// TIA Portal V16 export
// export: Created 2024-12-03T15:41:46.4557849Z, ExportSetting WithReadOnly, DisplayName Totally Integrated Automation Portal, DisplayVersion V16 Update 6, DisplayName TIA Portal Version Control Interface, DisplayVersion V16 Update 2, DisplayName TIA Portal Openness, DisplayVersion V16 Update 6, DisplayName TIA Portal Teamcenter Gateway, DisplayVersion V16, DisplayName SINAMICS Startdrive Advanced, DisplayVersion V16 Update 5, DisplayName SINAMICS Startdrive G130, G150, S120, S150, SINAMICS MV, S210, DisplayVersion V16 Update 5, DisplayName SINAMICS Startdrive G110M, G120, G120C, G120D, G120P, G115D, DisplayVersion V16 Update 5, DisplayName STEP 7 Professional, DisplayVersion V16 Update 6, DisplayName STEP 7 Safety, DisplayVersion V16, DisplayName WinCC Advanced / Unified PC, DisplayVersion V16 Update 6
TYPE "System_Counters_UDT"
// stored: CreationDate 2021-07-13T07:41:36.2278727Z, InterfaceModifiedDate 2021-03-11T07:33:04.7322472Z, IsConsistent true, LibraryConformanceStatus The object is library-conformant., ModifiedDate 2021-03-27T07:36:47.4918093Z
   STRUCT
      Infeed_1 : UInt;
      Infeed_2 : UInt;
      Infeed_3 : UInt;
      Infeed_4 : UInt;
      Infeed_5 : UInt;
      MainLane_Total : UInt;
      Scan100_Reject : UInt;
      Scan100_Exit1 : UInt;
      Scan100_Exit2 : UInt;
      Scan100MainLane : UInt;
      Scan200_Rejct : UInt;
      Scan200_Printer1 : UInt;
      Scan200_Printer2 : UInt;
      Scan200_Printer3 : UInt;
      Scan200_MainLane : UInt;
      MezzanineRetour_Printer1 : UInt;
      MezzanineRetour_Printer2 : UInt;
      Printer1_OK : UInt;
      Printer1_NOK : UInt;
      Printer2_OK : UInt;
      Printer2_NOK : UInt;
      Printer3_OK : UInt;
      Printer3_NOK : UInt;
   END_STRUCT;
END_TYPE
